FUNCTION_BLOCK FB_State2 EXTENDS FB_State
VAR_INPUT
END_VAR
VAR_OUTPUT
END_VAR
VAR
END_VAR

END_FUNCTION_BLOCK

(* stored: Version 1.1.0.1, ProductVersion 3.1.4024.12
   POU FB_State2: Id {337171c7-0d93-460d-abc6-c4886fad044c}, SpecialFunc None *)
